TYPE ST_SQLValue  :
STRUCT
    sValue : STRING(255);
END_STRUCT
END_TYPE

(* stored: Version 1.1.0.1, ProductVersion 3.1.4026.18
   DUT ST_SQLValue: Id {ba2326a1-0ddb-4346-bb8b-729de023295f} *)
